(* CoDeSys 2.3 library: TcBase.lib *)

(* Data type *)
TYPE
	FW_NoOfByte :
(
	NoOfByte_Byte	:=	1,
	NoOfByte_Word	:=	2,
	NoOfByte_DWord	:=	4
);
END_TYPE

(* Data type *)
TYPE FW_SystemInfoType
STRUCT
	runTimeNo				:	BYTE;
	projectName				:	STRING(32);
	numberOfTasks			:	BYTE;
	onlineChangeCount		:	UINT;
	bootDataFlags			:	BYTE;
	systemStateFlags		:	WORD;
END_STRUCT
END_TYPE

(* Data type *)
TYPE FW_SystemTaskInfoType
STRUCT
	active					:	BOOL;
	taskName				:	STRING(16);
	firstCycle				:	BOOL;
	cycleTimeExceeded		:	BOOL;
	cycleTime				:	UDINT;
	lastExecTime			:	UDINT;
	priority				:	BYTE;
	cycleCount				: 	UDINT;
END_STRUCT
END_TYPE

(* Data type *)
TYPE FW_TcEvent :
STRUCT
	Class 					: 	UDINT;
	Prio 					: 	UDINT;
	Id 						: 	UDINT;
	bQuitRequired 			: 	BOOL;
	DataFormatStrAddress 	: 	UDINT;
	UserFlags 				: 	DWORD;
	Flags 					: 	DWORD;
	StreamType 				: 	UDINT;
	SourceString 			: 	STRING[15];   		(* TCEVENT_SRCNAMESIZE *)
	SourceId 				: 	UDINT;
	ProgId 					:  	STRING[31];			(* TCEVENT_FMTPRGSIZE *)
END_STRUCT
END_TYPE

(* POU FW_AdsClearEvents, ST *)
FUNCTION_BLOCK FW_AdsClearEvents
VAR_INPUT
	sNetId				:	STRING(23);
	bClear 				: 	BOOL;
	nMode				:	UDINT;
	tTimeout			:	TIME;
END_VAR
VAR_OUTPUT
	bBusy				:	BOOL;
	bError				:	BOOL;
	nErrId				:	UDINT;
END_VAR
VAR
	STAMP_I				:	UINT;
	ACCESSCNT_I			:	UDINT;
	BUSY_I				:	BOOL;
	ERR_I				:	BOOL;
	ERRID_I				:	UDINT;
	READ_SAV_I			:	BOOL;
	TICKSTART_I			:	UDINT;
END_VAR
;
END_FUNCTION_BLOCK

(* POU FW_AdsLogDINT, ST *)
FUNCTION FW_AdsLogDINT : DINT
VAR_INPUT
	nCtrlMask		:	DWORD;
	sMsgFmt			:	STRING(255);
	nArg			:	DINT;
END_VAR
;
END_FUNCTION

(* POU FW_AdsLogEvent, ST *)
FUNCTION_BLOCK FW_AdsLogEvent
VAR_INPUT
	sNetId					:	STRING(23);
	nPort					:	UINT;
	bEvent					:	BOOL;
	bEventQuit				:	BOOL;
	stEventConfigData		:	FW_TcEvent;
	pEventDataAddress		:	UDINT;		(* pointer *)
	cbEventDataLength		:	UDINT;
	bFbCleanup				:	BOOL;
	tTimeout				:	TIME;
END_VAR
VAR_OUTPUT
	nEventState				:	UDINT;
	bError					:	BOOL;
	nErrId					:	UDINT;
	bQuit					:	BOOL;
END_VAR
VAR
	STAMPREQ_I				:	UINT;
	STAMPRES_I				:	UINT;
	STAMPSIG_I				:	UINT;
	STAMPCON_I				:	UINT;
	ACCESSCNT_I				:	UDINT;
	AMSADDR_I				:	ARRAY[1..8] OF BYTE;
	EVENT_I					:	FW_TcEvent ;
	pTCEVENTSTREAM_I		:	UDINT;
	CBEVENTSTREAM_I			:	UDINT;
	nSTATE_I				:	DINT;
	nSTATEREQ_I				:	DINT;
	nSTATERES_I				:	DINT;
	nSTATESIG_I				:	DINT;
	nSTATECON_I				:	DINT;
	ERR_I					:	BOOL;
	ERRID_I					:	UDINT;
	bEVENT_SAV_I			:	BOOL;
	bEVENTQUIT_SAV_I		:	BOOL;
	TICKSTART_I				:	UDINT;
END_VAR
;
END_FUNCTION_BLOCK

(* POU FW_AdsLogLREAL, ST *)
FUNCTION FW_AdsLogLREAL : DINT
VAR_INPUT
	nCtrlMask			:	DWORD;
	sMsgFmt				:	STRING(255);
	fArg				:	LREAL;
END_VAR
;
END_FUNCTION

(* POU FW_AdsLogSTR, ST *)
FUNCTION FW_AdsLogSTR 	: 	DINT
VAR_INPUT
	nCtrlMask			:	DWORD;
	sMsgFmt				:	STRING(255);
	sArg				:	STRING(255);
END_VAR
;
END_FUNCTION

(* POU FW_AdsRdWrt, ST *)
FUNCTION_BLOCK FW_AdsRdWrt
VAR_INPUT
	sNetId			:	STRING(23);
	nPort			:	UINT;
	nIdxGrp			:	UDINT;
	nIdxOffs		:	UDINT;
	cbWriteLen		:	UDINT;
	cbReadLen		:	UDINT;
	pWriteBuff 		:	DWORD;
	pReadBuff		:	DWORD;
	bExecute		:	BOOL;
	tTimeout		:	TIME;
END_VAR
VAR_OUTPUT
	bBusy			:	BOOL;
	bError			:	BOOL;
	nErrId			:	UDINT;
	cbRead			:	UDINT;				(* count of bytes actually read *)
END_VAR
VAR
	STAMP_I			:	UINT;
	ACCESSCNT_I		:	UDINT;
	BUSY_I			:	BOOL;
	ERR_I			:	BOOL;
	ERRID_I			:	UDINT;
	WRTRD_SAV_I		:	BOOL;
	PDESTADDR_I		:	DWORD;
	TICKSTART_I		:	UDINT;
END_VAR
;
END_FUNCTION_BLOCK

(* POU FW_AdsRdWrtInd, ST *)
FUNCTION_BLOCK FW_AdsRdWrtInd
VAR_INPUT
	bClear			:	BOOL;
END_VAR
VAR_OUTPUT
	bValid			: 	BOOL;
	sNetId			:	STRING(23);
	nPort			:	UINT;
	nInvokeId		:	UDINT;
	nIdxGrp			:	UDINT;
	nIdxOffs		:	UDINT;
	cbReadLen		:	UDINT;
	cbWriteLen		:	UDINT;
	pWriteBuff	 	:	DWORD;
END_VAR
VAR
	CLEAR_I			:	BOOL;
END_VAR
;
END_FUNCTION_BLOCK

(* POU FW_AdsRdWrtRes, ST *)
FUNCTION_BLOCK FW_AdsRdWrtRes
VAR_INPUT
	sNetId			:	STRING(23);
	nPort			:	UINT;
	nInvokeId		:	UDINT;
	nErrId			:	UDINT;
	cbReadLen		:	UDINT;
	pReadBuff		:	DWORD;
	bRespond		:	BOOL;
END_VAR
VAR_OUTPUT
END_VAR
VAR
	RESPOND_I		:	BOOL;
END_VAR
;
END_FUNCTION_BLOCK

(* POU FW_AdsRead, ST *)
FUNCTION_BLOCK FW_AdsRead
VAR_INPUT
	sNetId		:	STRING(23);
	nPort		:	UINT;
	nIdxGrp		:	UDINT;
	nIdxOffs	:	UDINT;
	cbReadLen	:	UDINT;
	pReadBuff	:	DWORD;
	bExecute	:	BOOL;
	tTimeout	:	TIME;
END_VAR
VAR_OUTPUT
	bBusy		:	BOOL;
	bError		:	BOOL;
	nErrId		:	UDINT;
	cbRead		:	UDINT;				(* count of bytes actually read *)
END_VAR
VAR
	STAMP_I		:	UINT;
	ACCESSCNT_I	:	UDINT;
	BUSY_I		:	BOOL;
	ERR_I		:	BOOL;
	ERRID_I		:	UDINT;
	READ_SAV_I	:	BOOL;
	TICKSTART_I	:	UDINT;
END_VAR
;
END_FUNCTION_BLOCK

(* POU FW_AdsReadDeviceInfo, ST *)
FUNCTION_BLOCK FW_AdsReadDeviceInfo
VAR_INPUT
	sNetId			:	STRING(23);
	nPort			:	UINT;
	bExecute		:	BOOL;
	tTimeout		:	TIME;
END_VAR
VAR_OUTPUT
	bBusy			:	BOOL;
	bError			:	BOOL;
	nErrId			:	UDINT;
	sDevName		:	STRING(19);
	nDevVersion		:	UDINT;
END_VAR
VAR
	STAMP_I			:	UINT;
	ACCESSCNT_I		:	UDINT;
	BUSY_I			:	BOOL;
	ERR_I			:	BOOL;
	ERRID_I			:	UDINT;
	RDINFO_SAV_I	:	BOOL;
	TICKSTART_I		:	UDINT;
END_VAR
;
END_FUNCTION_BLOCK

(* POU FW_AdsReadInd, ST *)
FUNCTION_BLOCK FW_AdsReadInd
VAR_INPUT
	bClear			:	BOOL;
END_VAR
VAR_OUTPUT
	bValid			: 	BOOL;
	sNetId			:	STRING(23);
	nPort			:	UINT;
	nInvokeId		:	UDINT;
	nIdxGrp			:	UDINT;
	nIdxOffs		:	UDINT;
	cbReadLen		:	UDINT;
END_VAR
VAR
	CLEAR_I		:	BOOL;
END_VAR
;
END_FUNCTION_BLOCK

(* POU FW_AdsReadRes, ST *)
FUNCTION_BLOCK FW_AdsReadRes
VAR_INPUT
	sNetId			:	STRING(23);
	nPort			:	UINT;
	nInvokeId		:	UDINT;
	nErrId			:	UDINT;
	cbReadLen		:	UDINT;
	pReadBuff		:	DWORD;
	bRespond		:	BOOL;
END_VAR
VAR_OUTPUT
END_VAR
VAR
	RESPOND_I		:	BOOL;
END_VAR
;
END_FUNCTION_BLOCK

(* POU FW_AdsReadState, ST *)
FUNCTION_BLOCK FW_AdsReadState
VAR_INPUT
	sNetId			:	STRING(23);
	nPort			:	UINT;
	bExecute		:	BOOL;
	tTimeout		:	TIME;
END_VAR
VAR_OUTPUT
	bBusy			:	BOOL;
	bError			:	BOOL;
	nErrId			:	UDINT;
	nAdsState		:	UINT;
	nDevState		:	UINT;
END_VAR
VAR
	STAMP_I			:	UINT;
	ACCESSCNT_I		:	UDINT;
	BUSY_I			:	BOOL;
	ERR_I			:	BOOL;
	ERRID_I			:	UDINT;
	RDSTATE_SAV_I	:	BOOL;
	TICKSTART_I		:	UDINT;
END_VAR
;
END_FUNCTION_BLOCK

(* POU FW_AdsWrite, ST *)
FUNCTION_BLOCK FW_AdsWrite
VAR_INPUT
	sNetId		:	STRING(23);
	nPort		:	UINT;
	nIdxGrp		:	UDINT;
	nIdxOffs	:	UDINT;
	cbWriteLen	:	UDINT;
	pWriteBuff 	:	DWORD;
	bExecute	:	BOOL;
	tTimeout	:	TIME;
END_VAR
VAR_OUTPUT
	bBusy		:	BOOL;
	bError		:	BOOL;
	nErrId		:	UDINT;
END_VAR
VAR
	STAMP_I		:	UINT;
	ACCESSCNT_I:	UDINT;
	BUSY_I		:	BOOL;
	ERR_I		:	BOOL;
	ERRID_I		:	UDINT;
	WRITE_SAV_I	:	BOOL;
	TICKSTART_I	:	UDINT;
END_VAR
;
END_FUNCTION_BLOCK

(* POU FW_AdsWriteControl, ST *)
FUNCTION_BLOCK FW_AdsWriteControl
VAR_INPUT
	sNetId			:	STRING(23);
	nPort			:	UINT;
	nAdsState		:	UINT;
	nDevState		:	UINT;
	cbWriteLen		:	UDINT;
	pWriteBuff	 	:	DWORD;
	bExecute		:	BOOL;
	tTimeout		:	TIME;
END_VAR
VAR_OUTPUT
	bBusy			:	BOOL;
	bError			:	BOOL;
	nErrId			:	UDINT;
END_VAR
VAR
	STAMP_I			:	UINT;
	ACCESSCNT_I		:	UDINT;
	BUSY_I			:	BOOL;
	ERR_I			:	BOOL;
	ERRID_I			:	UDINT;
	WRITE_SAV_I		:	BOOL;
	TICKSTART_I		:	UDINT;
END_VAR
;
END_FUNCTION_BLOCK

(* POU FW_AdsWriteInd, ST *)
FUNCTION_BLOCK FW_AdsWriteInd
VAR_INPUT
	bClear			:	BOOL;
END_VAR
VAR_OUTPUT
	bValid			: 	BOOL;
	sNetId			:	STRING(23);
	nPort			:	UINT;
	nInvokeId		:	UDINT;
	nIdxGrp			:	UDINT;
	nIdxOffs		:	UDINT;
	cbWriteLen		:	UDINT;
	pWriteBuff	 	:	DWORD;
END_VAR
VAR
	CLEAR_I			:	BOOL;
END_VAR
;
END_FUNCTION_BLOCK

(* POU FW_AdsWriteRes, ST *)
FUNCTION_BLOCK FW_AdsWriteRes
VAR_INPUT
	sNetId			:	STRING(23);
	nPort			:	UINT;
	nInvokeId		:	UDINT;
	nErrId			:	UDINT;
	bRespond		:	BOOL;
END_VAR
VAR_OUTPUT
END_VAR
VAR
	RESPOND_I		:	BOOL;
END_VAR
;
END_FUNCTION_BLOCK

(* POU FW_DRand, ST *)
FUNCTION_BLOCK FW_DRand
VAR_INPUT
	nSeed			:	INT;
END_VAR
VAR_OUTPUT
	fRndNum			:	LREAL;
END_VAR
VAR
	FirstCall_i		:	BOOL;
	HoldRand_i		:	DINT;
	R250_Buffer_i	:	ARRAY[0..249] OF UINT;
	R250_Index		:	INT;
END_VAR
;
END_FUNCTION_BLOCK

(* POU FW_GetCpuAccount, ST *)
FUNCTION_BLOCK FW_GetCpuAccount
VAR_INPUT
END_VAR
VAR_OUTPUT
	dwCpuAccount	:	UDINT;
END_VAR
;
END_FUNCTION_BLOCK

(* POU FW_GetCpuCounter, ST *)
FUNCTION_BLOCK FW_GetCpuCounter
VAR_INPUT
END_VAR
VAR_OUTPUT
	dwCpuCntLo	:	UDINT;
	dwCpuCntHi	:	UDINT;
END_VAR
;
END_FUNCTION_BLOCK

(* POU FW_GetCurTaskIndex, ST *)
FUNCTION_BLOCK FW_GetCurTaskIndex
VAR_INPUT
END_VAR
VAR_OUTPUT
	nIndex: BYTE;
END_VAR
;
END_FUNCTION_BLOCK

(* POU FW_GetSystemTime, ST *)
FUNCTION_BLOCK FW_GetSystemTime
VAR_INPUT
END_VAR
VAR_OUTPUT
	dwTimeLo	:	UDINT;
	dwTimeHi	:	UDINT;
END_VAR
VAR
END_VAR
;
END_FUNCTION_BLOCK

(* POU FW_GetVersionTcBase, ST *)
FUNCTION FW_GetVersionTcBase : 	UINT	(*Gets the library version info *)
VAR_INPUT
	nVersionElement				:	INT;
END_VAR
(*
	Possible nVersionElement parameter:
	1	:	major number
	2	:	minor number
	3	:	revision number
*)
VAR
END_VAR
(* Version history:
Date          	| Version    	| created under      		| Author          		| Remark 
------------------------------------------------------------------------------------------------------------------------------------------------------- 
01.10.2001    	| 1.0.0	      	| V2.8.0 (Build 707) 		| Christoph C.     	| first release 
07.10.2002    	| 1.0.1      		| V2.8.0 (Build 735) 		| Christoph C.     	| FW_MemMove function added
03.05.2004	| 1.0.2		| V2.9.0 (Build 959)		| JP				| FW_PortRead, FW_PortWrite new		
21.11.2004	| 1.0.3		| V2.10.0 (Build 1243)	| Christoph C.		| F_GetVersionTcBase fix. Branched version of TcBase.lib (for TwinCAT 2.9 and TwinCAT 2.10 builds only)
06.06.2006	| 1.0.4		| V2.10.0 (Build 1257)	| Christoph C.		| FW_PortWrite returns FALSE if running on other CPU than X86
30.04.2009	| 1.0.5		| V2.11.0 (Build 1522)	| Christoph C.		| New Internal (firmware) function/fb: FW_CallGenericFun, FW_CallGenericFb
14.05.2009	| 1.0.6		| V2.11.0 (Build 1524)	| Christoph C.		| New generic firmware function added: F_GetCurDcTaskTime
*) 
;
END_FUNCTION

(* POU FW_LptSignal, ST *)
FUNCTION FW_LptSignal : BOOL
(*
	This function allows the control of the data output pins on the line printer connector.
	It can be used for time measurement purposes with a hardware oscilloscope.
*) 
VAR_INPUT
	nPortAddr 	:	UINT;
	nPinNo		: 	UINT;
	bOnOff		:	BOOL;
END_VAR
;
END_FUNCTION

(* POU FW_MemCmp, ST *)
FUNCTION FW_MemCmp 	: 	DINT	(* Compare characters in two buffers. *)
VAR_INPUT
	pBuf1			:	UDINT;	(* First buffer *)
	pBuf2			:	UDINT;	(* Second buffer *)
	cbLen			:	UDINT;	(* Number of characters *)
END_VAR
(*
	Return value: 
		=	-1 	: 	buf1 less than buf2 
		= 	0 	: 	buf1 identical to buf2 
		=	1 	:	buf1 greater than buf2 
		= 	255	:	Error (pBuf1 = 0 OR pBuf2 = 0 OR cbLen = 0 )	
*)
VAR
END_VAR
;
END_FUNCTION

(* POU FW_MemCpy, ST *)
FUNCTION FW_MemCpy 	: 	UDINT	(* Copies characters between buffers. *)
VAR_INPUT
	pDest			:	UDINT;	(* New buffer *)
	pSrc			:	UDINT;	(* Buffer to copy from *)
	cbLen			:	UDINT;	(* Number of characters to copy *)
END_VAR
(*
	Return value: 
		> 0	:	The number succesfully copied bytes 
		= 0	:	Error ( pDest = 0 OR pSrc = 0 OR cbLen = 0 )	
*)

VAR
END_VAR
;
END_FUNCTION

(* POU FW_MemMove, ST *)
(* 	Copies characters between buffers. If some regions of the source area and the destination overlap,
	FW_MemMove ensures that the original source bytes in the overlapping region are copied before being overwritten. *)
FUNCTION FW_MemMove 	: 	UDINT
VAR_INPUT
	pDest			:	UDINT;	(* New buffer *)
	pSrc			:	UDINT;	(* Buffer to copy from *)
	cbLen			:	UDINT;	(* Number of characters to copy *)
END_VAR
(*
	Return value: 
		> 0	:	The number succesfully copied bytes 
		= 0	:	Error ( pDest = 0 OR pSrc = 0 OR cbLen = 0 )	
*)

VAR
END_VAR
;
END_FUNCTION

(* POU FW_MemSet, ST *)
FUNCTION FW_MemSet 	: 	UDINT	(* Sets buffers to a specified character. *)
VAR_INPUT
	pDest			:	UDINT;	(* Pointer to destination *)
	nFillByte		:	USINT;	(* Character to set *)
	cbLen			:	UDINT;	(* Number of characters *)
END_VAR
(*
	Return value: 
		> 0	:	The number of set bytes 
		= 0	:	Error ( pDest = 0 OR cbLen = 0 )	
*)

VAR
END_VAR
;
END_FUNCTION

(* POU FW_PortRead, ST *)
FUNCTION FW_PortRead : DWORD
(*
	This function allows to read a port.
*) 
VAR_INPUT
	nPortAddr 	:	UDINT;
	eNoOfByte	: 	FW_NoOfByte;
END_VAR
;
END_FUNCTION

(* POU FW_PortWrite, ST *)
FUNCTION FW_PortWrite : BOOL
(*
	This function allows to write a port.
*) 
VAR_INPUT
	nPortAddr 	:	UDINT;
	eNoOfByte	: 	FW_NoOfByte ;
	nValue		:	DWORD;
END_VAR
;
END_FUNCTION
